// TwinCAT 3 PLC project TcoRexrothPressTests
// Title: TcoRexrothPressTests
// Company: Vortex.Library
// ProjectVersion: 0.6.0.913
// ProgramVersion: 3.1.4024.12
// libraries:
//   Tc2_Standard, * (Beckhoff Automation GmbH)
//   Tc2_System, * (Beckhoff Automation GmbH)
//   Tc3_Module, * (Beckhoff Automation GmbH)
//   TcoAbstractions, 0.6.0.913 (Vortex.Library)
//   TcoCognexVision, 0.6.0.913 (Vortex.Library)
//   TcoCore, 0.6.0.913 (Vortex.Library)
//   TcoIo, 0.6.0.913 (Vortex.Library)
//   TcoRexrothPress, 0.6.0.913 (Vortex.Library)
//   TcoUtilities, 0.6.0.913 (Vortex.Library)
// project tree:
//   GVLs/ GVL.TcGVL, GVL_iXlinker.TcGVL
//   / PlcTask.TcTTO
//   POUs/ MAIN.TcPOU, TcoContext.TcPOU
// (motion and I/O tree: see PLC project tcorexrothpress)
// real-time tasks:
//   TASK PlcTask: cycle T#10ms, priority 20, ADS port 350
//   TASK PNIO: cycle T#16ms, priority 21, ADS port 351
//   TASK PlcTask1: cycle T#10ms, priority 22, ADS port 352
// variable links:
//   TcoRexrothPressTests/TcoRexrothPressTests Instance <-> Device 1 (EtherCAT)/Press (IndraDrive MPC20 (1 CCD Master +0 CCD Slaves))
//     PlcTask Inputs/GVL_iXlinker.AdsAddr/netId <-> InfoData/AdsAddr/netId
//     PlcTask Inputs/GVL_iXlinker.AdsAddr/port <-> InfoData/AdsAddr/port
//     PlcTask Inputs/GVL_iXlinker.RexrothPress.Response.DigitalIoMapping <-> AT (CCD Master)/PLC output WORD8 AT %QB16
//     PlcTask Inputs/GVL_iXlinker.RexrothPress.Response.Handle <-> AT (CCD Master)/PLC output WORD4 AT %QB8
//     PlcTask Inputs/GVL_iXlinker.RexrothPress.Response.NotificationForce <-> AT (CCD Master)/PLC Global Register A24
//     PlcTask Inputs/GVL_iXlinker.RexrothPress.Response.NotificationId <-> AT (CCD Master)/PLC output WORD6 AT %QB12
//     PlcTask Inputs/GVL_iXlinker.RexrothPress.Response.NotificationPosition <-> AT (CCD Master)/Position feedback value 1
//     PlcTask Inputs/GVL_iXlinker.RexrothPress.Response.NotificationStatus <-> AT (CCD Master)/PLC output WORD7 AT %QB14
//     PlcTask Inputs/GVL_iXlinker.RexrothPress.Response.NotificationValue <-> AT (CCD Master)/PLC Global Register A23
//     PlcTask Inputs/GVL_iXlinker.RexrothPress.Response.NotificationVelocity <-> AT (CCD Master)/Velocity feedback value of encoder 1
//     PlcTask Inputs/GVL_iXlinker.RexrothPress.Response.Status <-> AT (CCD Master)/PLC output WORD5 AT %QB10
//     PlcTask Inputs/GVL_iXlinker.RexrothPress.Response.Value1 <-> AT (CCD Master)/PLC Global Register A20
//     PlcTask Inputs/GVL_iXlinker.RexrothPress.Response.Value2 <-> AT (CCD Master)/PLC Global Register A22
//     PlcTask Inputs/GVL_iXlinker.RexrothPress.Response.Value3 <-> AT (CCD Master)/PLC Global Register A21
//     PlcTask Inputs/GVL_iXlinker.RexrothPress.Response.VirtualIo <-> AT (CCD Master)/PLC output WORD9 AT %QB18
//     PlcTask Outputs/GVL_iXlinker.RexrothPress.Request.Command <-> MDT (CCD Master)/PLC input WORD5 AT %IB10
//     PlcTask Outputs/GVL_iXlinker.RexrothPress.Request.Handle <-> MDT (CCD Master)/PLC input WORD4 AT %IB8
//     PlcTask Outputs/GVL_iXlinker.RexrothPress.Request.Value1 <-> MDT (CCD Master)/PLC Global Register A17
//     PlcTask Outputs/GVL_iXlinker.RexrothPress.Request.Value2 <-> MDT (CCD Master)/PLC Global Register A18
//     PlcTask Outputs/GVL_iXlinker.RexrothPress.Request.Value3 <-> MDT (CCD Master)/PLC Global Register A19
//     PlcTask Outputs/GVL_iXlinker.RexrothPress.Request.Value7 <-> MDT (CCD Master)/PLC Global Register A25
//     PlcTask Outputs/GVL_iXlinker.RexrothPress.Request.Value4 <-> MDT (CCD Master)/PLC Global Register A4
//     PlcTask Outputs/GVL_iXlinker.RexrothPress.Request.Value5 <-> MDT (CCD Master)/PLC Global Register A5
//     PlcTask Outputs/GVL_iXlinker.RexrothPress.Request.Value6 <-> MDT (CCD Master)/PLC Global Register A6
//     PlcTask Outputs/GVL_iXlinker.RexrothPress.Request.VirtualIo <-> MDT (CCD Master)/PLC input WORD6 AT %IB12

CONFIGURATION TcoRexrothPressTests
    RESOURCE PLC ON TwinCAT3
        TASK PlcTask(INTERVAL := T#16ms, PRIORITY := 21);
        PROGRAM MAIN WITH PlcTask : MAIN;
    END_RESOURCE
END_CONFIGURATION

// ---- GVLs/GVL.TcGVL
{attribute 'qualified_only'}
VAR_GLOBAL
END_VAR

// ---- GVLs/GVL_iXlinker.TcGVL
{attribute 'qualified_only'}
VAR_GLOBAL
    {attribute addProperty Name "Press IO"}
    RexrothPress : TcoSmartFunctionKitIO_v_4_x_x;
    {attribute addProperty Name "AdsAddr"}
    AdsAddr AT %I* : TcoAmsAddr;
    {attribute addProperty Name "State"}
    State AT %I* : UINT;
END_VAR

// ---- POUs/MAIN.TcPOU
PROGRAM MAIN
VAR
    myVeryFirstTcoContextInstance : TcoContext;
END_VAR

myVeryFirstTcoContextInstance.Run();

END_PROGRAM

// ---- POUs/TcoContext.TcPOU
FUNCTION_BLOCK TcoContext EXTENDS TcoCore.TcoContext
VAR
    {attribute addProperty Name "<#My very first SFK#>"}
    sfk : TcoRexrothPress.TcoSmartFunctionKit_v_4_x_x(THIS^);
END_VAR

(*~
    <docu>
        <summary>
            Main method of the TcoContext. This is the entry point of any control logic that belongs to this context.
            The call of this method is ensured by calling the <c>InstanceName.Run()</c> method, and it must not be called explicitly.
            This method is abstract, and it must be overridden in derived block.
        </summary>
    </docu>
~*)
METHOD PROTECTED Main
VAR
    adsInfo : AMSADDR;
END_VAR
Sfk.Config.ErrorTime := T#20S;
Sfk.Config.InfoTime := T#10S;
sfk.Config.CurveExportLocation := 'd:\expot\'; // if empty export not performed
sfk.Config.IpAddress := '192.168.0.1'; // for rest comunication
adsInfo.netId := GVL_iXlinker.AdsAddr.netId; //ads info from eCAT bus
adsInfo.port := GVL_iXlinker.AdsAddr.port;
sfk(inoIoData := GVL_iXlinker.RexrothPress, AdsAddr := adsInfo);
sfk.Service();
END_METHOD

END_FUNCTION_BLOCK
